// TIA Portal V20 export
TYPE "LER_typePartStatus"
// stored: Access Published
   STRUCT
      partPresent { ExternalWritable := 'False'} : Bool;   // 검사 하기 전 제품 있음
      partEnabled { ExternalWritable := 'False'} : Bool;   // 검사 결과 ok
      partDisabled { ExternalWritable := 'False'} : Bool;   // 검사 결과 ng
      inspectionPart { ExternalWritable := 'False'} : Bool;   // 검사 전
      masterPart { ExternalWritable := 'False'} : Bool;   // 검사기 캘리용 마스터 샘플
      status5 { ExternalWritable := 'False'} : Bool;   // Spare
      dummyPart { ExternalWritable := 'False'} : Bool;   // 더미 데이터
      partDryRun { ExternalWritable := 'False'} : Bool;   // 공운전 데이터
   END_STRUCT;
END_TYPE
